# EPICS StreamDevice protocol: Stream/photo.proto
terminator = CR LF;

id {
	ExtraInput = Ignore;
	out "ID?";
	in "%100c";
}

photo {
	out "PHO:?";
	in "%d";
}

debug{
	ExtraInput = Ignore;
        out "%s";
        in "%39c";
}
